// TIA Portal V20 export
VAR_GLOBAL   // PLC tag table "00_Simulation"
   "AAxxxSP1.Slot1.I.16" AT %I1.0 : Bool;   // SIMIT Simulation currently running (life bit from SIMIT, always TRUE while SIMIT is running)
END_VAR
